(* Schneider Machine Expert - Basic project SAU2, file version 2.0.0.0 *)
(* ProjectInformations: Name=New project *)

HARDWARE
  Cpu 0: TM221CE16T
  Cartridge1 0: TMC2SL1
  EthernetConfiguration: NetworkName=M221, IpAllocationMode=FixedAddress, IpAddress=192.168.1.12, SubnetMask=255.255.255.0
  EthernetConfiguration: NetworkName=M221, IpAllocationMode=FixedAddress, IpAddress=0.0.0.0, SubnetMask=0.0.0.0
  SerialLineConfiguration: Baud=Baud9600, Parity=ParityNone, DataBits=DataBits8, StopBits=StopBits1, PhysicalMedium=PhysicalMediumRs485, TransmissionMode=TransmissionModeModbusRtu, SlaveId=1, Addressing=MasterAddressing
  MastTask: UsePeriodScanMode=false, PeriodScan=100
  FastTask: Period=255
  CpuBehavior: StartingMode=StartAsPreviousState, AutoSaveRamOnEeprom=true, WatchdogPeriod=250

SYMBOLS  (address, symbol, comment, settings)
  %S5       SB_TB100MS  "内部时钟生成的 100 毫秒时基"
  %TM0        [Preset=15, Base=OneSecond]
  %TM1        [Preset=10, Base=TenMilliSeconds]
  %TM2        [Preset=15, Base=OneSecond]
  %TM3        [Preset=15, Base=OneSecond]
  %TM4        [Preset=15, Base=OneSecond]
  %TM5        [Preset=15, Base=OneSecond]
  %TM6        [Preset=15, Base=OneSecond]
  %TM7        [Preset=15, Base=OneSecond]
  %READ_VAR0   [Link(Value(FBComLinkParameterEnums=SerialLine1)), RemoteDeviceId(Value(int=1)), Timeout(Value(int=3)), ObjType(Value(FBComObjTypeParameterEnums=IW)), FirstObj(Value(int=513)), Quantity(Value(int=4)), IndexData(Value(int=0))]
  %READ_VAR1   [Link(Value(FBComLinkParameterEnums=SerialLine1)), RemoteDeviceId(Value(int=2)), Timeout(Value(int=3)), ObjType(Value(FBComObjTypeParameterEnums=IW)), FirstObj(Value(int=513)), Quantity(Value(int=11)), IndexData(Value(int=10))]
  %READ_VAR2   [Link(Value(FBComLinkParameterEnums=SerialLine1)), RemoteDeviceId(Value(int=3)), Timeout(Value(int=3)), ObjType(Value(FBComObjTypeParameterEnums=IW)), FirstObj(Value(int=513)), Quantity(Value(int=11)), IndexData(Value(int=30))]
  %READ_VAR3   [Link(Value(FBComLinkParameterEnums=SerialLine1)), RemoteDeviceId(Value(int=4)), Timeout(Value(int=3)), ObjType(Value(FBComObjTypeParameterEnums=IW)), FirstObj(Value(int=513)), Quantity(Value(int=8)), IndexData(Value(int=50))]
  %READ_VAR4   [Link(Value(FBComLinkParameterEnums=SerialLine1)), RemoteDeviceId(Value(int=5)), Timeout(Value(int=3)), ObjType(Value(FBComObjTypeParameterEnums=IW)), FirstObj(Value(int=513)), Quantity(Value(int=8)), IndexData(Value(int=60))]
  %READ_VAR5   [Link(Value(FBComLinkParameterEnums=SerialLine1)), RemoteDeviceId(Value(int=6)), Timeout(Value(int=3)), ObjType(Value(FBComObjTypeParameterEnums=IW)), FirstObj(Value(int=513)), Quantity(Value(int=8)), IndexData(Value(int=70))]
  %READ_VAR6   [Link(Value(FBComLinkParameterEnums=SerialLine1)), RemoteDeviceId(Value(int=7)), Timeout(Value(int=3)), ObjType(Value(FBComObjTypeParameterEnums=IW)), FirstObj(Value(int=513)), Quantity(Value(int=8)), IndexData(Value(int=80))]
  %READ_VAR7   [Link(Value(FBComLinkParameterEnums=SerialLine1)), RemoteDeviceId(Value(int=2)), Timeout(Value(int=3)), ObjType(Value(FBComObjTypeParameterEnums=IW)), FirstObj(Value(int=536)), Quantity(Value(int=1)), IndexData(Value(int=25))]
  %READ_VAR8   [Link(Value(FBComLinkParameterEnums=SerialLine1)), RemoteDeviceId(Value(int=3)), Timeout(Value(int=3)), ObjType(Value(FBComObjTypeParameterEnums=IW)), FirstObj(Value(int=536)), Quantity(Value(int=1)), IndexData(Value(int=45))]

POU Communication
  (* SectionNumber=0 *)

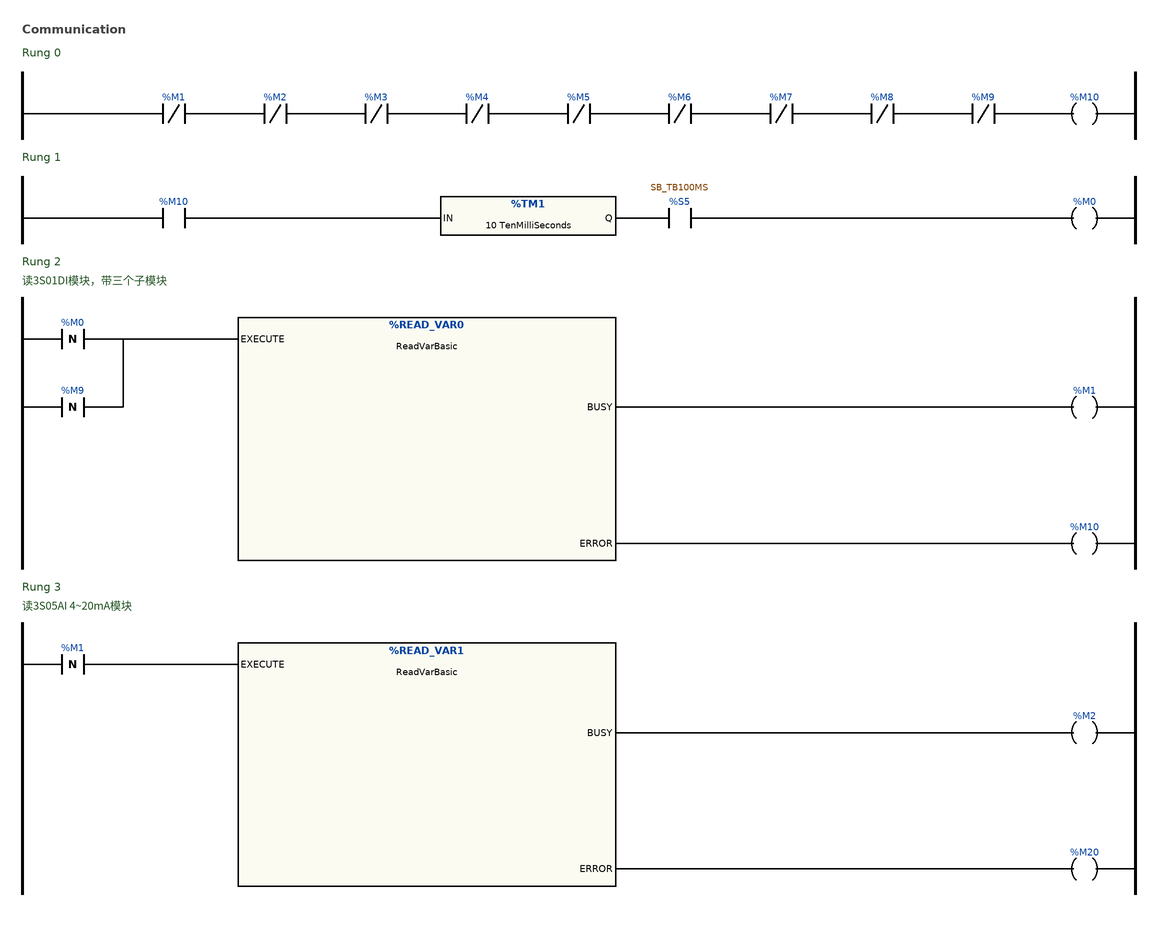

// Rung 0
  LDN %M1
  ANDN %M2
  ANDN %M3
  ANDN %M4
  ANDN %M5
  ANDN %M6
  ANDN %M7
  ANDN %M8
  ANDN %M9
  ST %M10
  // as ST:
  //   %M10 := NOT %M1 AND NOT %M2 AND NOT %M3 AND NOT %M4 AND NOT %M5 AND NOT %M6 AND NOT %M7 AND NOT %M8 AND NOT %M9;

// Rung 1
  BLK %TM1
  LD %M10
  IN
  OUT_BLK
  LD Q
  AND %S5                 (* SB_TB100MS *)
  ST %M0
  END_BLK
  // as ST:
  //   %TM1(IN := %M10);
  //   %M0 := %TM1.Q AND SB_TB100MS;

// Rung 2
// 读3S01DI模块，带三个子模块
  BLK %READ_VAR0
  LDF %M0
  ORF %M9
  EXECUTE
  OUT_BLK
  LD BUSY
  ST %M1
  LD ERROR
  ST %M10
  END_BLK
  // as ST:
  //   %READ_VAR0(EXECUTE := FALLING(%M0) OR FALLING(%M9));
  //   %M1 := %READ_VAR0.BUSY;
  //   %M10 := %READ_VAR0.ERROR;

// Rung 3
// 读3S05AI 4~20mA模块
  BLK %READ_VAR1
  LDF %M1
  EXECUTE
  OUT_BLK
  LD BUSY
  ST %M2
  LD ERROR
  ST %M20
  END_BLK
  // as ST:
  //   %READ_VAR1(EXECUTE := FALLING(%M1));
  //   %M2 := %READ_VAR1.BUSY;
  //   %M20 := %READ_VAR1.ERROR;

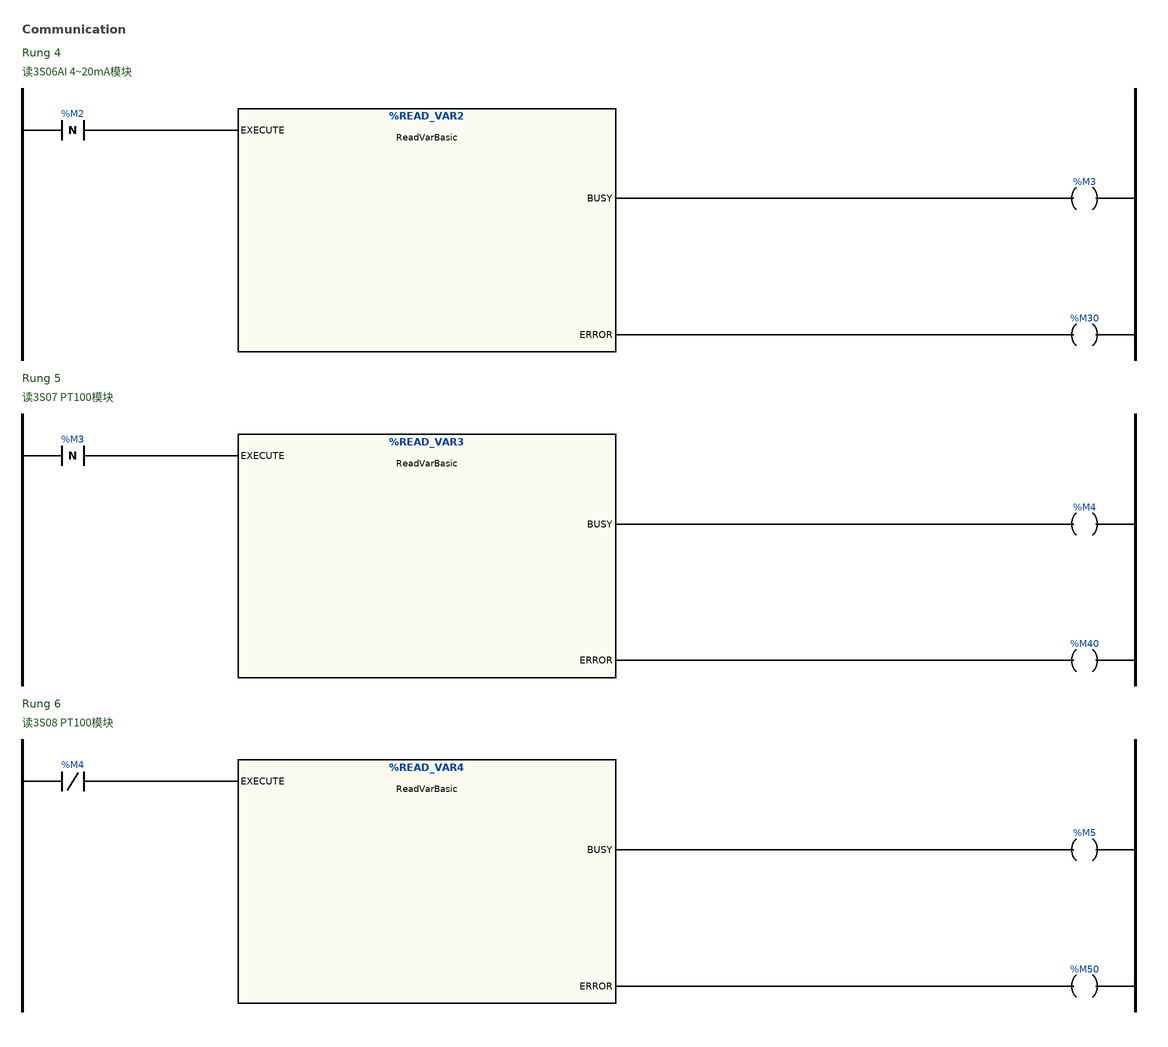

// Rung 4
// 读3S06AI 4~20mA模块
  BLK %READ_VAR2
  LDF %M2
  EXECUTE
  OUT_BLK
  LD BUSY
  ST %M3
  LD ERROR
  ST %M30
  END_BLK
  // as ST:
  //   %READ_VAR2(EXECUTE := FALLING(%M2));
  //   %M3 := %READ_VAR2.BUSY;
  //   %M30 := %READ_VAR2.ERROR;

// Rung 5
// 读3S07 PT100模块
  BLK %READ_VAR3
  LDF %M3
  EXECUTE
  OUT_BLK
  LD BUSY
  ST %M4
  LD ERROR
  ST %M40
  END_BLK
  // as ST:
  //   %READ_VAR3(EXECUTE := FALLING(%M3));
  //   %M4 := %READ_VAR3.BUSY;
  //   %M40 := %READ_VAR3.ERROR;

// Rung 6
// 读3S08 PT100模块
  BLK %READ_VAR4
  LDN %M4
  EXECUTE
  OUT_BLK
  LD BUSY
  ST %M5
  LD ERROR
  ST %M50
  END_BLK
  // as ST:
  //   %READ_VAR4(EXECUTE := NOT %M4);
  //   %M5 := %READ_VAR4.BUSY;
  //   %M50 := %READ_VAR4.ERROR;

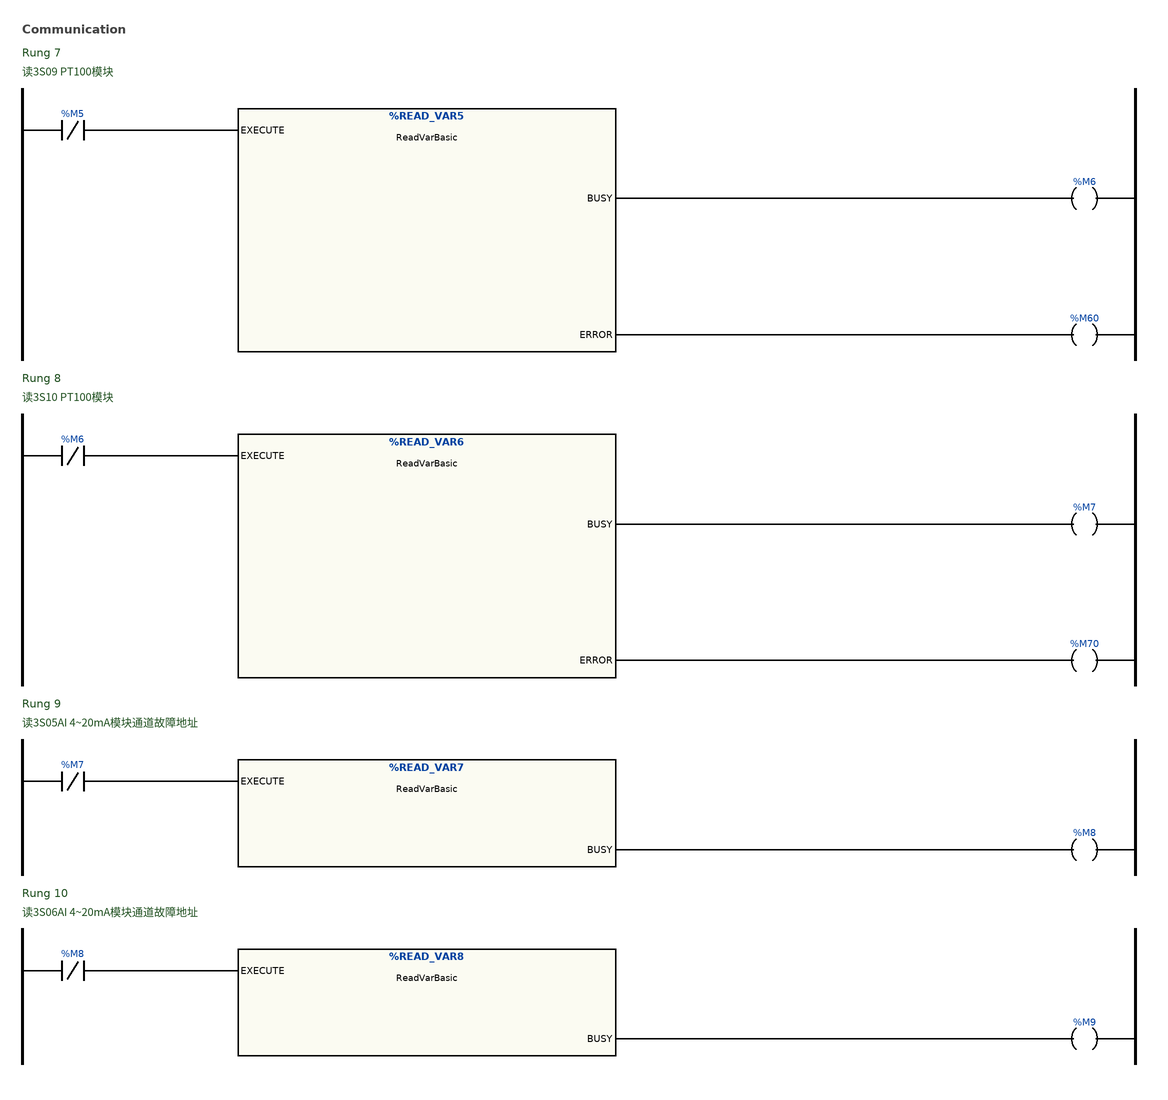

// Rung 7
// 读3S09 PT100模块
  BLK %READ_VAR5
  LDN %M5
  EXECUTE
  OUT_BLK
  LD BUSY
  ST %M6
  LD ERROR
  ST %M60
  END_BLK
  // as ST:
  //   %READ_VAR5(EXECUTE := NOT %M5);
  //   %M6 := %READ_VAR5.BUSY;
  //   %M60 := %READ_VAR5.ERROR;

// Rung 8
// 读3S10 PT100模块
  BLK %READ_VAR6
  LDN %M6
  EXECUTE
  OUT_BLK
  LD BUSY
  ST %M7
  LD ERROR
  ST %M70
  END_BLK
  // as ST:
  //   %READ_VAR6(EXECUTE := NOT %M6);
  //   %M7 := %READ_VAR6.BUSY;
  //   %M70 := %READ_VAR6.ERROR;

// Rung 9
// 读3S05AI 4~20mA模块通道故障地址
  BLK %READ_VAR7
  LDN %M7
  EXECUTE
  OUT_BLK
  LD BUSY
  ST %M8
  END_BLK
  // as ST:
  //   %READ_VAR7(EXECUTE := NOT %M7);
  //   %M8 := %READ_VAR7.BUSY;

// Rung 10
// 读3S06AI 4~20mA模块通道故障地址
  BLK %READ_VAR8
  LDN %M8
  EXECUTE
  OUT_BLK
  LD BUSY
  ST %M9
  END_BLK
  // as ST:
  //   %READ_VAR8(EXECUTE := NOT %M8);
  //   %M9 := %READ_VAR8.BUSY;

POU CommError
  (* SectionNumber=0 *)

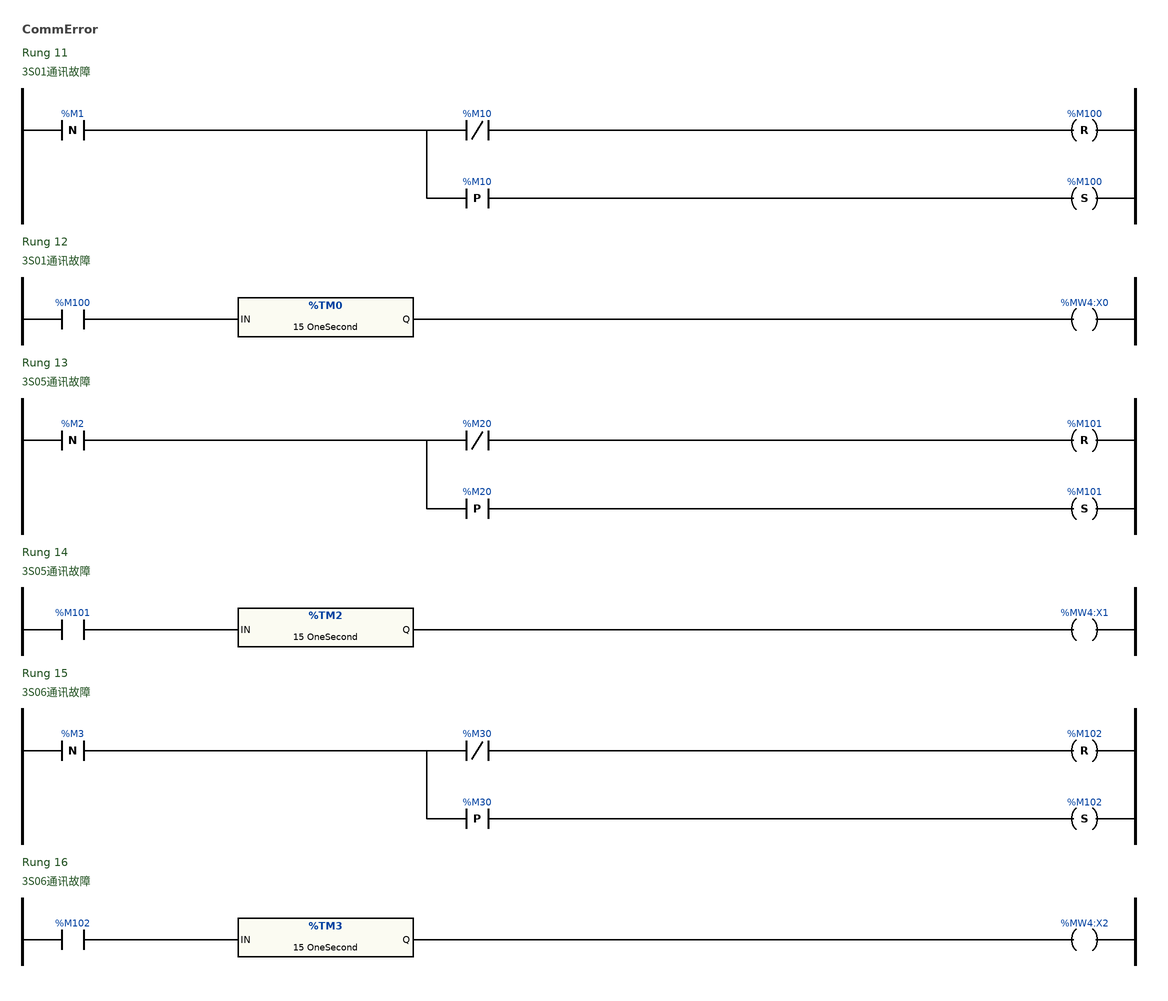

// Rung 11
// 3S01通讯故障
  LDF %M1
  MPS
  ANDN %M10
  R %M100
  MPP
  ANDR %M10
  S %M100
  // as ST:
  //   IF FALLING(%M1) AND NOT %M10 THEN %M100 := FALSE; END_IF;
  //   IF FALLING(%M1) AND RISING(%M10) THEN %M100 := TRUE; END_IF;

// Rung 12
// 3S01通讯故障
  BLK %TM0
  LD %M100
  IN
  OUT_BLK
  LD Q
  ST %MW4:X0
  END_BLK
  // as ST:
  //   %TM0(IN := %M100);
  //   %MW4:X0 := %TM0.Q;

// Rung 13
// 3S05通讯故障
  LDF %M2
  MPS
  ANDN %M20
  R %M101
  MPP
  ANDR %M20
  S %M101
  // as ST:
  //   IF FALLING(%M2) AND NOT %M20 THEN %M101 := FALSE; END_IF;
  //   IF FALLING(%M2) AND RISING(%M20) THEN %M101 := TRUE; END_IF;

// Rung 14
// 3S05通讯故障
  BLK %TM2
  LD %M101
  IN
  OUT_BLK
  LD Q
  ST %MW4:X1
  END_BLK
  // as ST:
  //   %TM2(IN := %M101);
  //   %MW4:X1 := %TM2.Q;

// Rung 15
// 3S06通讯故障
  LDF %M3
  MPS
  ANDN %M30
  R %M102
  MPP
  ANDR %M30
  S %M102
  // as ST:
  //   IF FALLING(%M3) AND NOT %M30 THEN %M102 := FALSE; END_IF;
  //   IF FALLING(%M3) AND RISING(%M30) THEN %M102 := TRUE; END_IF;

// Rung 16
// 3S06通讯故障
  BLK %TM3
  LD %M102
  IN
  OUT_BLK
  LD Q
  ST %MW4:X2
  END_BLK
  // as ST:
  //   %TM3(IN := %M102);
  //   %MW4:X2 := %TM3.Q;

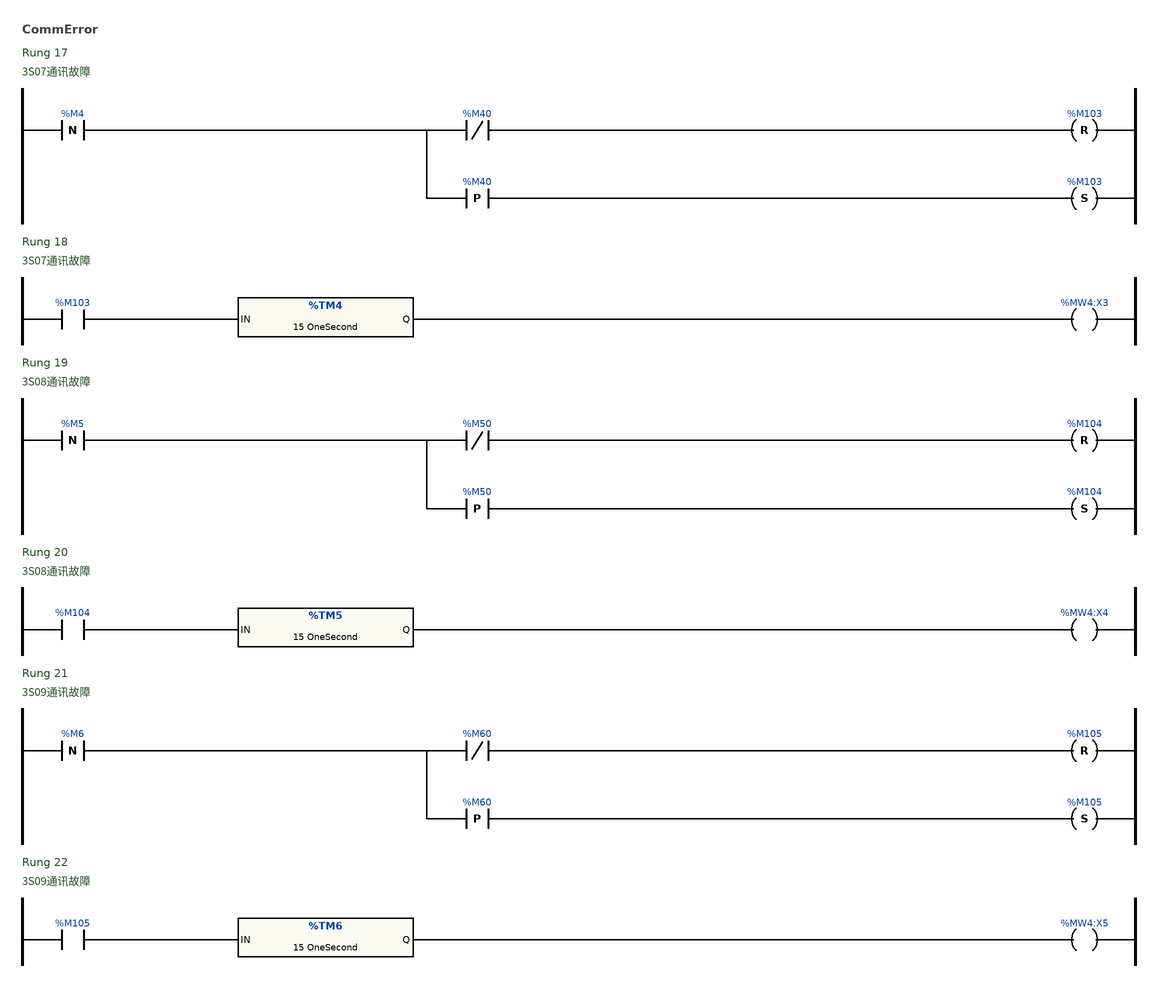

// Rung 17
// 3S07通讯故障
  LDF %M4
  MPS
  ANDN %M40
  R %M103
  MPP
  ANDR %M40
  S %M103
  // as ST:
  //   IF FALLING(%M4) AND NOT %M40 THEN %M103 := FALSE; END_IF;
  //   IF FALLING(%M4) AND RISING(%M40) THEN %M103 := TRUE; END_IF;

// Rung 18
// 3S07通讯故障
  BLK %TM4
  LD %M103
  IN
  OUT_BLK
  LD Q
  ST %MW4:X3
  END_BLK
  // as ST:
  //   %TM4(IN := %M103);
  //   %MW4:X3 := %TM4.Q;

// Rung 19
// 3S08通讯故障
  LDF %M5
  MPS
  ANDN %M50
  R %M104
  MPP
  ANDR %M50
  S %M104
  // as ST:
  //   IF FALLING(%M5) AND NOT %M50 THEN %M104 := FALSE; END_IF;
  //   IF FALLING(%M5) AND RISING(%M50) THEN %M104 := TRUE; END_IF;

// Rung 20
// 3S08通讯故障
  BLK %TM5
  LD %M104
  IN
  OUT_BLK
  LD Q
  ST %MW4:X4
  END_BLK
  // as ST:
  //   %TM5(IN := %M104);
  //   %MW4:X4 := %TM5.Q;

// Rung 21
// 3S09通讯故障
  LDF %M6
  MPS
  ANDN %M60
  R %M105
  MPP
  ANDR %M60
  S %M105
  // as ST:
  //   IF FALLING(%M6) AND NOT %M60 THEN %M105 := FALSE; END_IF;
  //   IF FALLING(%M6) AND RISING(%M60) THEN %M105 := TRUE; END_IF;

// Rung 22
// 3S09通讯故障
  BLK %TM6
  LD %M105
  IN
  OUT_BLK
  LD Q
  ST %MW4:X5
  END_BLK
  // as ST:
  //   %TM6(IN := %M105);
  //   %MW4:X5 := %TM6.Q;

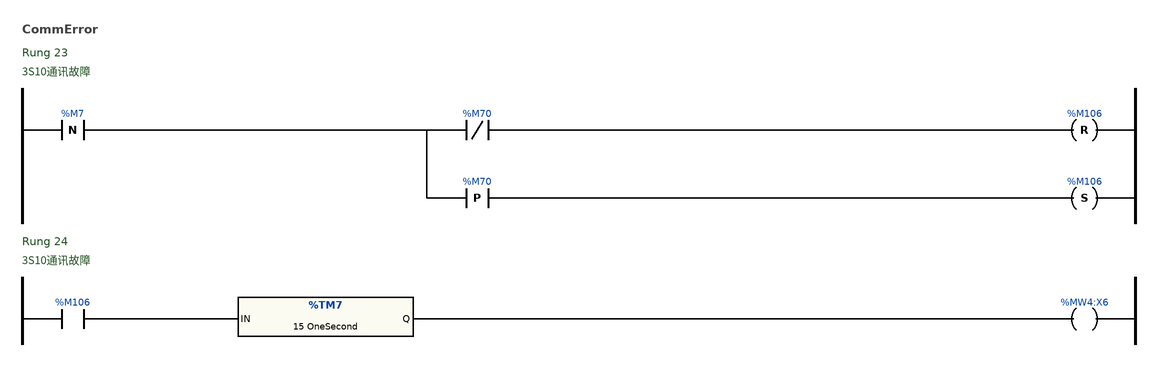

// Rung 23
// 3S10通讯故障
  LDF %M7
  MPS
  ANDN %M70
  R %M106
  MPP
  ANDR %M70
  S %M106
  // as ST:
  //   IF FALLING(%M7) AND NOT %M70 THEN %M106 := FALSE; END_IF;
  //   IF FALLING(%M7) AND RISING(%M70) THEN %M106 := TRUE; END_IF;

// Rung 24
// 3S10通讯故障
  BLK %TM7
  LD %M106
  IN
  OUT_BLK
  LD Q
  ST %MW4:X6
  END_BLK
  // as ST:
  //   %TM7(IN := %M106);
  //   %MW4:X6 := %TM7.Q;
